// Writes an sint32 value, without a tag, to the stream.
FUNCTION F_WriteSInt32 : HRESULT
VAR_IN_OUT
    aBuffer : ARRAY [*] OF BYTE;
    stState : ST_WriterInternalState;
END_VAR
VAR_INPUT
    nValue : DINT;
END_VAR
VAR
    nTmp : UDINT;
END_VAR

nTmp := F_EncodeZigZag32(nValue);
F_WriteSInt32 := F_WriteRawVarint32(aBuffer, stState, nTmp);

END_FUNCTION

(* stored: Version 1.1.0.1
   POU F_WriteSInt32: Id {01b4ad30-e64a-466f-9b41-61d0b834a634}, SpecialFunc None *)
